{attribute 'GeneratedUsingTerminal: EL9185--0000'}
{attribute addProperty BoxType "EL9185--0000"}
{attribute addProperty Description "EL9185 Potential Connection, 4 x 24-230V"}
{attribute addProperty Physics "KK"}
{attribute addProperty Id "EL9185"}
{attribute addProperty CRC "2630903271"}
{attribute addProperty Size "0"}
TYPE EL9185_9CD065E7 EXTENDS EtcSlaveTerminalBase_947E5A46 :
STRUCT
END_STRUCT
END_TYPE

(* stored: Version 1.2.0.0, ProductVersion 3.1.4024.11
   DUT EL9185_9CD065E7: Id {6c2f876d-d19c-41a1-8577-0ddbfee6ee68} *)
